PROGRAM prgPersistent
VAR
	fbUSV		: FB_WritePersistentData_CX81xx;

	fb_Reboot		: NT_reboot;
	m_Reboot		: BOOL:=FALSE;

END_VAR

fbUSV(
	eSaveModeData:= eUSVSaveMode.eSaveWhenPowerfail, 
	bLoadPersistentDataOk=> , 
	bPowerFailDetect=> , 
	bError=> , 
	bySaveProcess=> , 
	dwStorageLast24h=> , 
	udiErrorCode=> );
	
	
		
fb_Reboot(	netid := '',
			delay := 2,
			start := m_Reboot);

END_PROGRAM

(* stored: Version 1.1.0.1, ProductVersion 3.1.4024.11
   POU prgPersistent: Id {108c7acc-615a-428d-9d84-0b842341dda8}, SpecialFunc None *)
